// SIMATIC S7-200 project (STEP 7-Micro/WIN), CPU 224 REL 02.01

ORGANIZATION_BLOCK Briquette_Press_B_41:OB1
TITLE=B V4.1
// Custom program for WEIMA TH Standard Series briquette press.
//  #NVJOB Nicholas Veselov (independent developer) - https://nvjob.pro, http://nvjob.dx.am
// 
// ---------------------------------------------------------------------
// 
// INPUTS
// I0.0 - Power.
// I0.1 - Start the program in automatic mode.
// I0.2 - Stop the program in automatic mode.
// I0.3 - Manual mode.
// I0.4 - Vertical piston, sensor, lower position.
// I0.5 - Vertical piston, sensor, upper position.
// I0.6 - Horizontal piston, sensor, position retracted.
// I0.7 - Horizontal piston, sensor, position extended.
// I1.0 - Not involved.
// I1.1 - Valve button.
// I1.2 - Accident, stop.
// I1.3 - Change in operating time of the screw. Min time*.
// I1.4 - Change in the operating time of the screw. Max. time*.
// I1.5 - Not involved.
// 
// ---------------------------------------------------------------------
// 
// OUTPUTS
// Q0.0 - The engine of the hydraulic power station (star-delta).
// Q0.1 - Hydroelectric power station engine (star-delta).
// Q0.2 - Fan.
// Q0.3 - Auger.
// Q0.4 - Vertical piston, valve, up position (pushes down).
// Q0.5 - Vertical piston, valve, lower position (pushes up).
// Q0.6 - Horizontal piston, valve, retracts the piston.
// Q0.7 - Horizontal piston, valve, extends the piston.
// Q1.0 - Collet Piston.
// Q1.1 - Light Bulb Start
// 
BEGIN
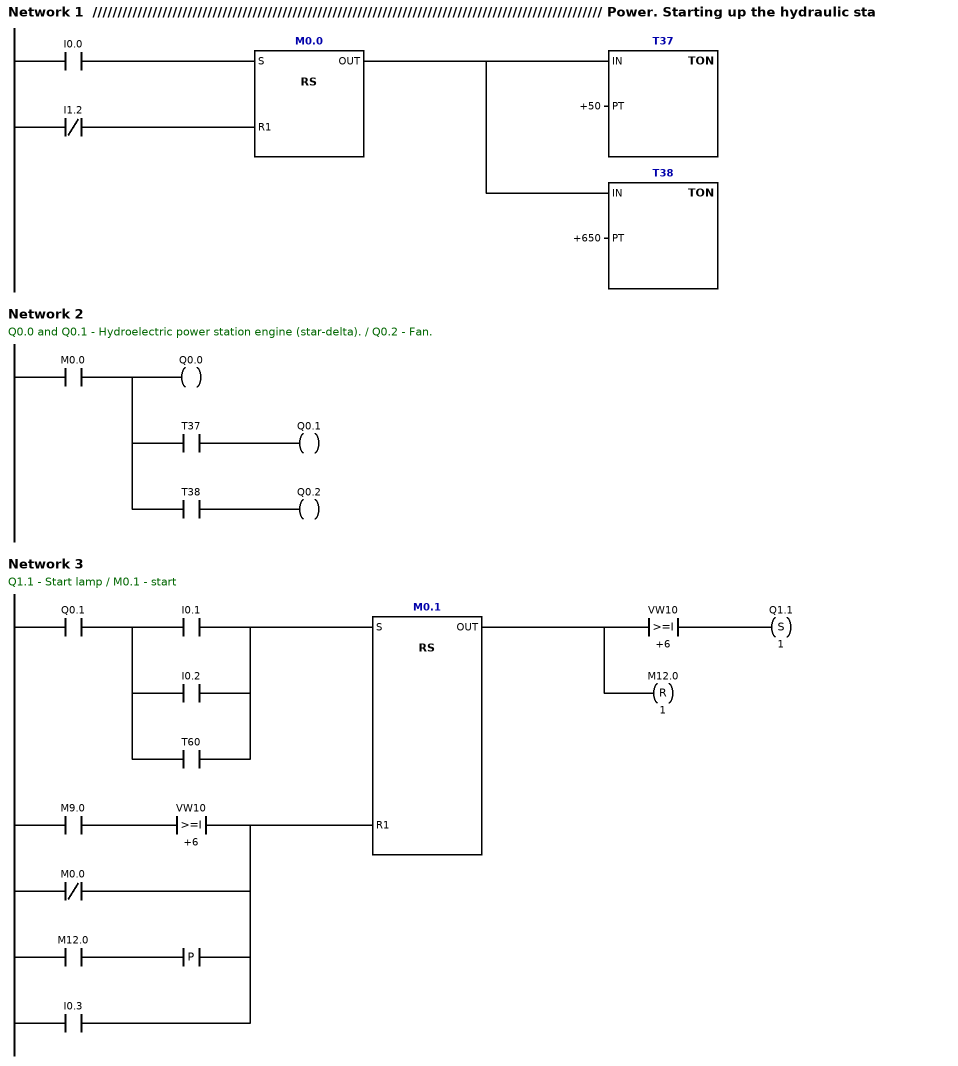
Network 1 // //////////////////////////////////////////////////////////////////////////////////////////////////////
Power. Starting up the hydraulic station.
//////////////////////////////////////////////////////////////////////////////////////////////////////
LD     I0.0
LDN    I1.2
NOT
LPS
A      M0.0
=      M0.0
LPP
ALD
O      M0.0
=      M0.0
TON    T37, +50
TON    T38, +650
Network 2
// Q0.0 and Q0.1 - Hydroelectric power station engine (star-delta).
// Q0.2 - Fan.
LD     M0.0
LPS
=      Q0.0
A      T37
=      Q0.1
LPP
A      T38
=      Q0.2
Network 3
// Q1.1 - Start lamp
// M0.1 - start
// (network saved uncompiled; LAD cells follow)
// row 0: c0 -| |- Q0.1 v  c1 -| |- I0.1 v  c2 --  c3 [RS M0.1 S:=power@row0, R1:=power@row3, OUT=>power]  c4 -- v  c5 -|>=I|- VW10, +6  c6 -(S) Q1.1, 1
// row 1: c0 ^v  c1 -| |- I0.2 ^v  c3 [box]  c4 ^  c5 -(R) M12.0, 1
// row 2: c0 ^  c1 -| |- T60 ^  c3 [box]
// row 3: c0 -| |- M9.0  c1 -|>=I|- VW10, +6 v  c2 --  c3 [box]
// row 4: c0 -|/|- M0.0  c1 -- ^v
// row 5: c0 -| |- M12.0  c1 -|P|-  ^v
// row 6: c0 -| |- I0.3  c1 -- ^
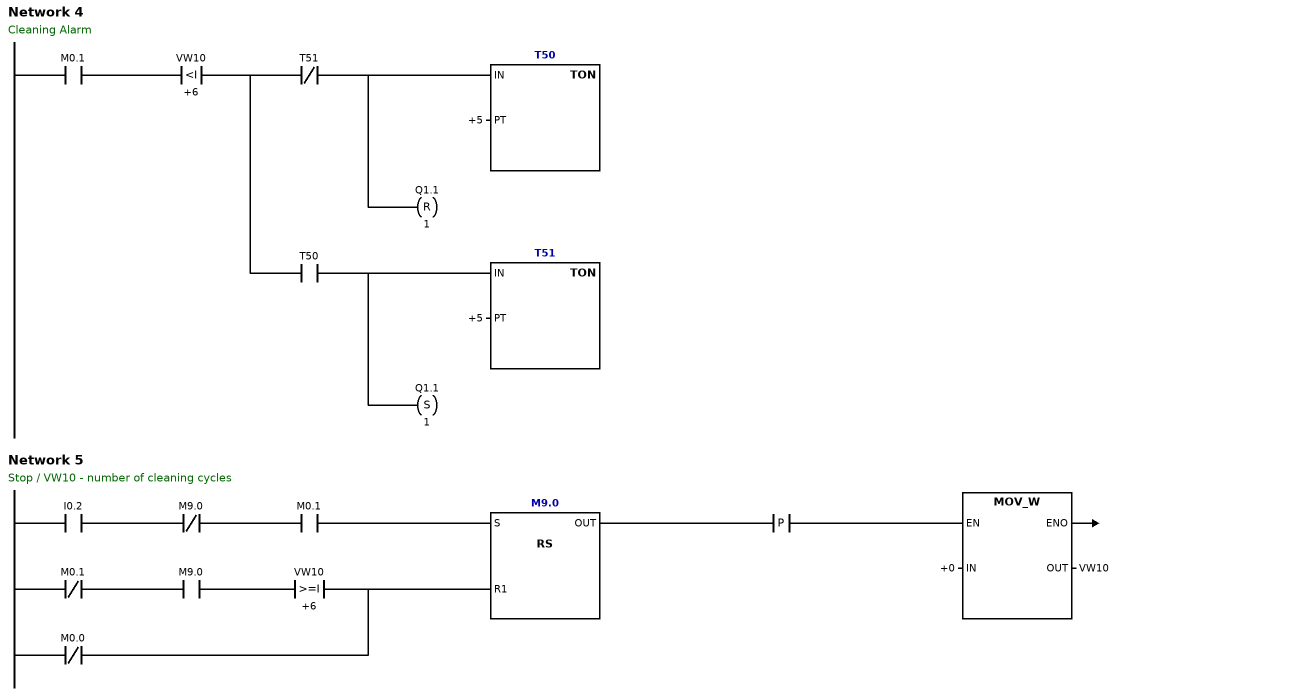
Network 4
// Cleaning Alarm
// (network saved uncompiled; LAD cells follow)
// row 0: c0 -| |- M0.1  c1 -|<I|- VW10, +6 v  c2 -|/|- T51 v  c3 --  c4 [TON T50 IN:=power@row0, PT:=+5]
// row 1: c1 ^v  c2 ^v  c4 [box]
// row 2: c1 ^v  c2 ^  c3 -(R) Q1.1, 1
// row 3: c1 ^  c2 -| |- T50 v  c3 --  c4 [TON T51 IN:=power@row3, PT:=+5]
// row 4: c2 ^v  c4 [box]
// row 5: c2 ^  c3 -(S) Q1.1, 1
Network 5
// Stop
// VW10 - number of cleaning cycles
// (network saved uncompiled; LAD cells follow)
// row 0: c0 -| |- I0.2  c1 -|/|- M9.0  c2 -| |- M0.1  c3 --  c4 [RS M9.0 S:=power@row0, R1:=power@row1, OUT=>power]  c5 --  c6 -|P|-  c7 --  c8 [MOV_W EN:=power@row0, IN:=+0, ENO=>power, OUT=>VW10]  c9 ->
// row 1: c0 -|/|- M0.1  c1 -| |- M9.0  c2 -|>=I|- VW10, +6 v  c3 --  c4 [box]  c8 [box]
// row 2: c0 -|/|- M0.0  c1 --  c2 -- ^
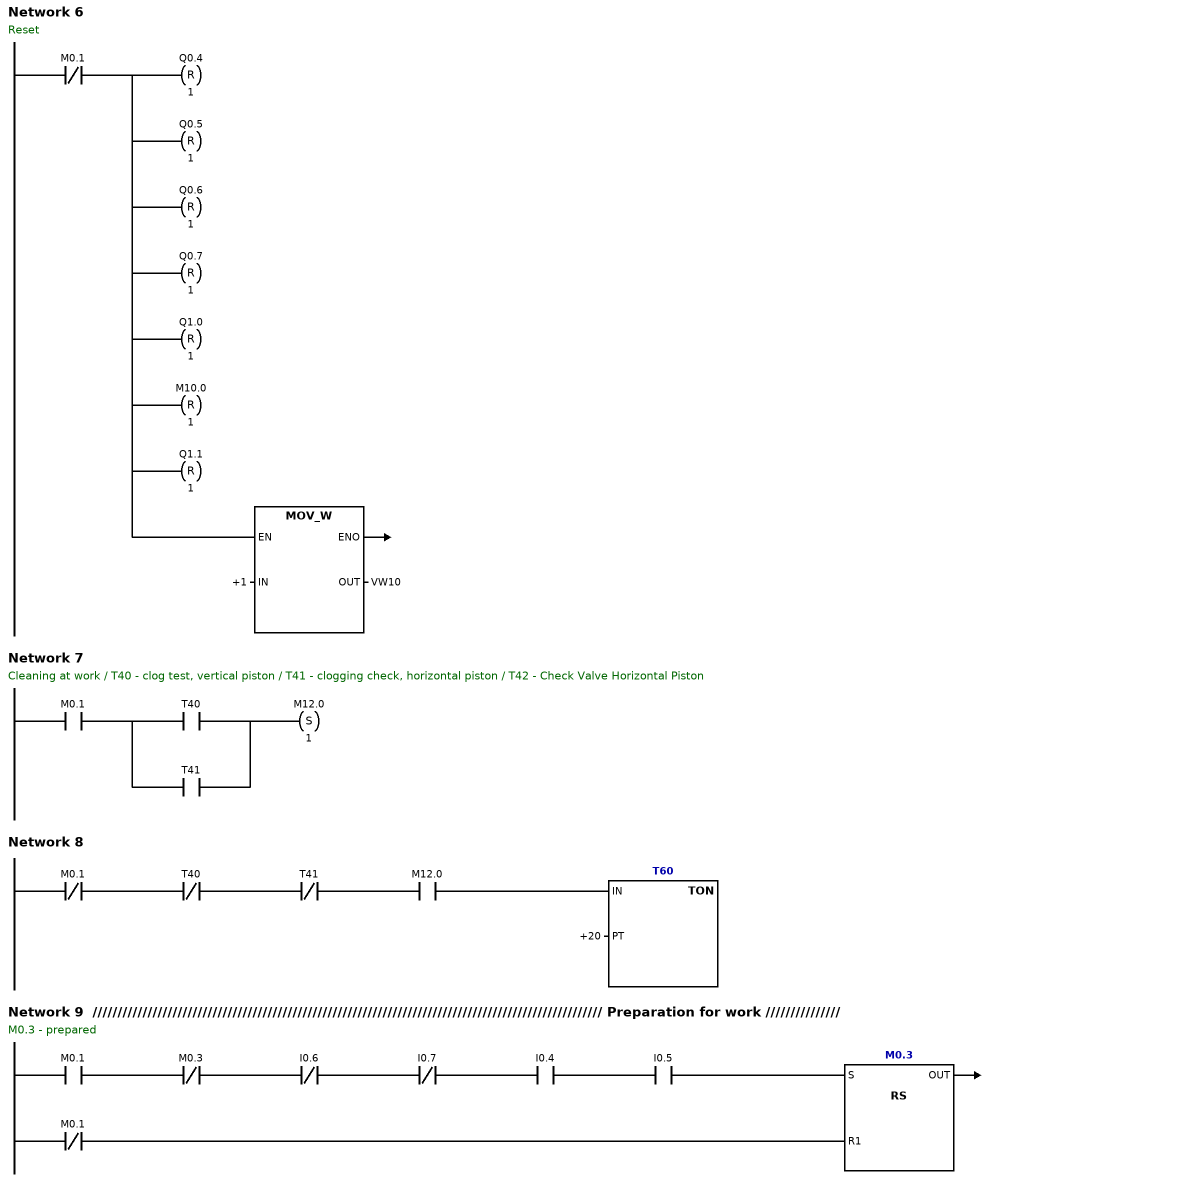
Network 6
// Reset
LDN    M0.1
R      Q0.4, 1
R      Q0.5, 1
R      Q0.6, 1
R      Q0.7, 1
R      Q1.0, 1
R      M10.0, 1
R      Q1.1, 1
MOVW   +1, VW10
Network 7
// Cleaning at work
// T40 - clog test, vertical piston
// T41 - clogging check, horizontal piston
// T42 - Check Valve Horizontal Piston
LD     M0.1
LD     T40
O      T41
ALD
S      M12.0, 1
Network 8
LDN    M0.1
AN     T40
AN     T41
A      M12.0
TON    T60, +20
Network 9 // //////////////////////////////////////////////////////////////////////////////////////////////////////
Preparation for work
//////////////////////////////////////////////////////////////////////////////////////////////////////
// M0.3 - prepared
LD     M0.1
AN     M0.3
AN     I0.6
AN     I0.7
A      I0.4
A      I0.5
LDN    M0.1
NOT
LPS
A      M0.3
=      M0.3
LPP
ALD
O      M0.3
=      M0.3
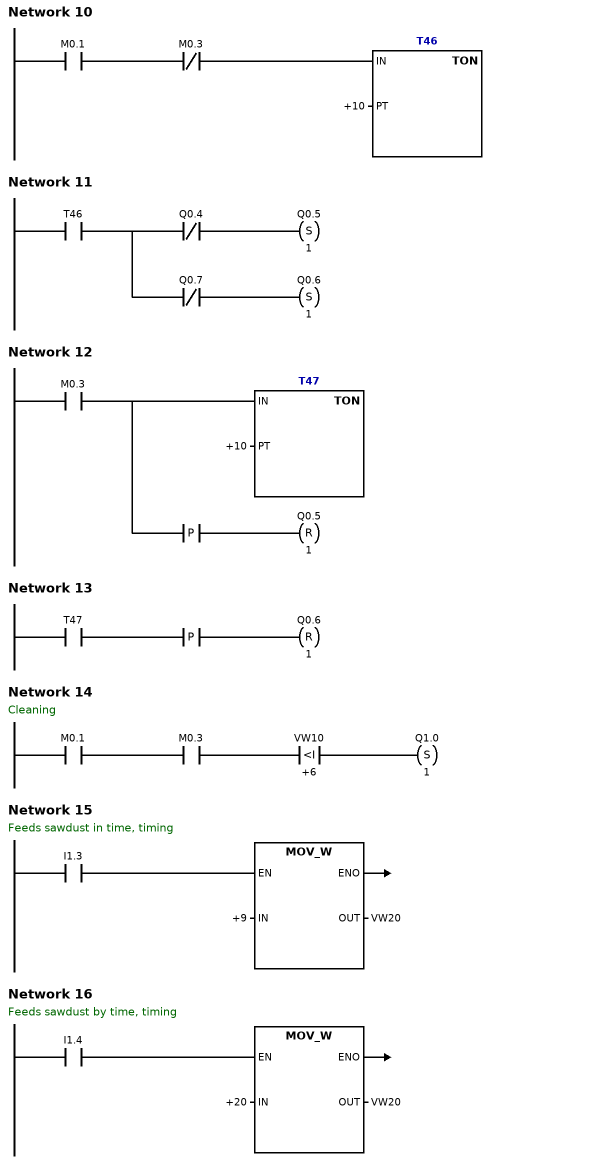
Network 10
LD     M0.1
AN     M0.3
TON    T46, +10
Network 11
LD     T46
LPS
AN     Q0.4
S      Q0.5, 1
LPP
AN     Q0.7
S      Q0.6, 1
Network 12
LD     M0.3
TON    T47, +10
EU
R      Q0.5, 1
Network 13
LD     T47
EU
R      Q0.6, 1
Network 14
// Cleaning
// (network saved uncompiled; LAD cells follow)
// row 0: c0 -| |- M0.1  c1 -| |- M0.3  c2 -|<I|- VW10, +6  c3 -(S) Q1.0, 1
Network 15
// Feeds sawdust in time, timing
LD     I1.3
MOVW   +9, VW20
Network 16
// Feeds sawdust by time, timing
LD     I1.4
MOVW   +20, VW20
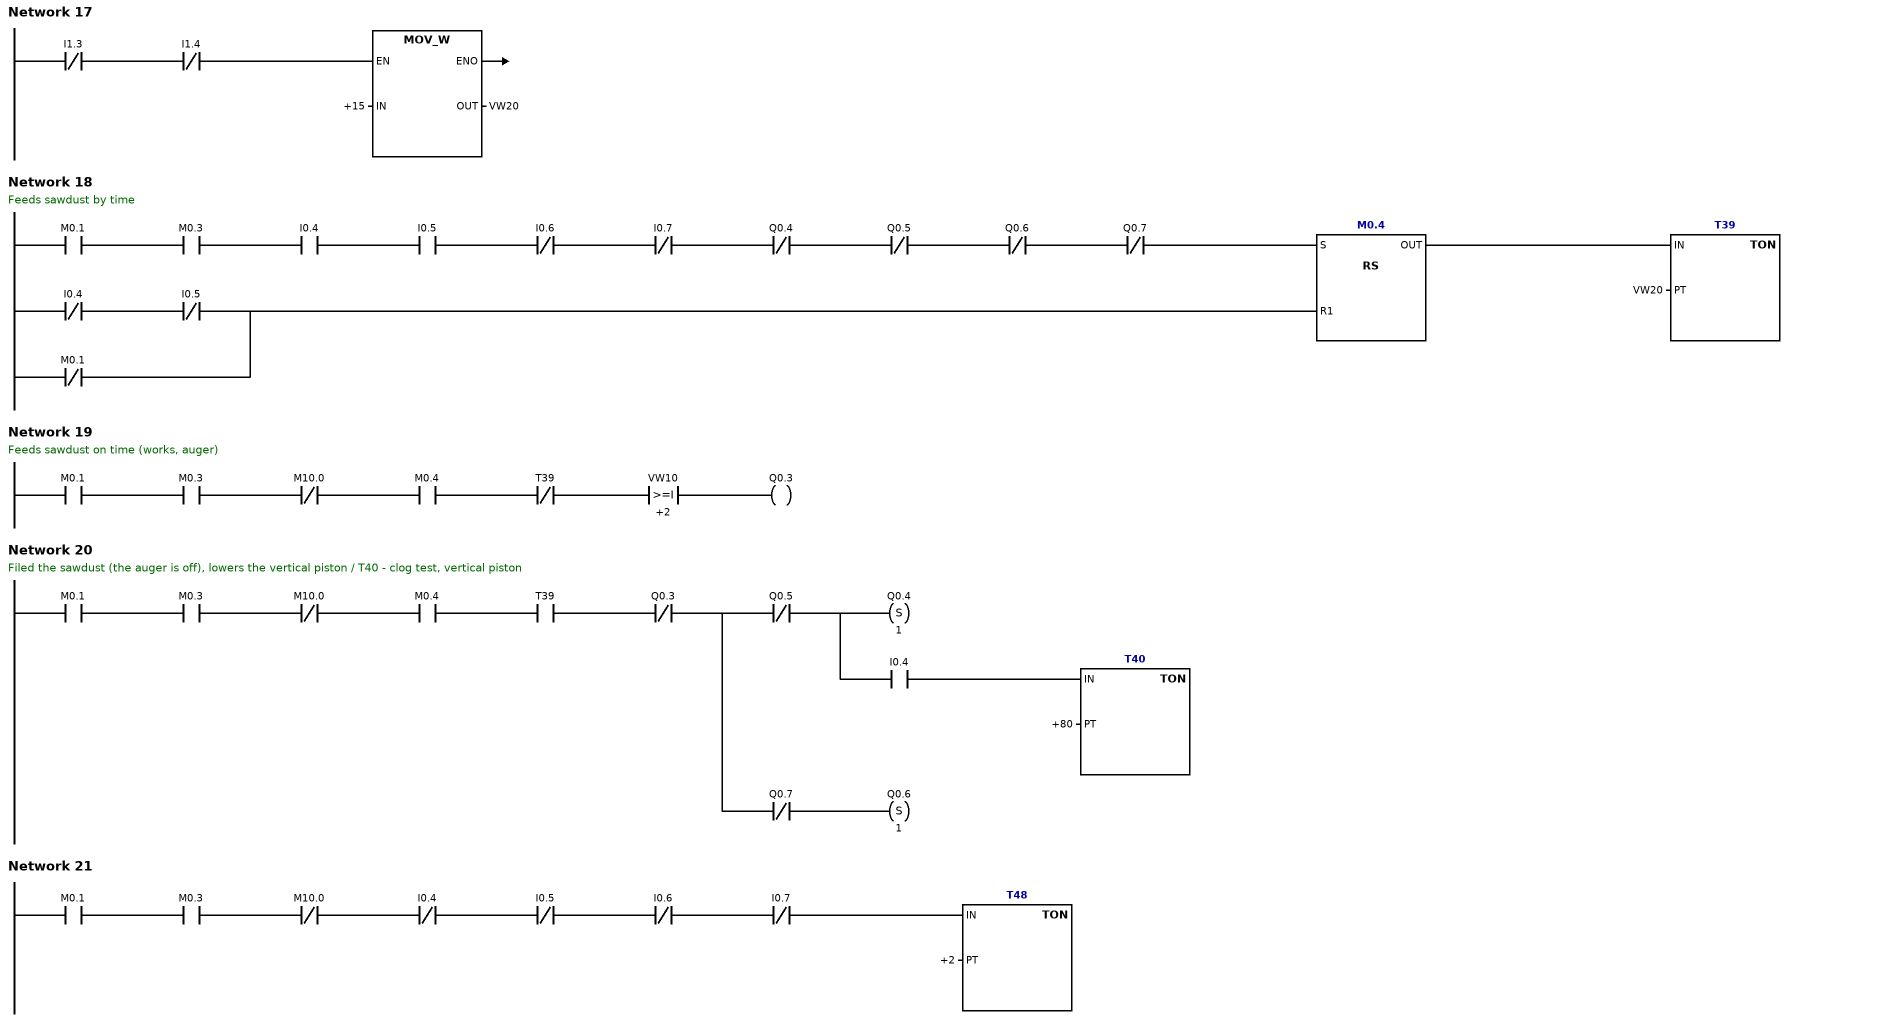
Network 17
LDN    I1.3
AN     I1.4
MOVW   +15, VW20
Network 18
// Feeds sawdust by time
LD     M0.1
A      M0.3
A      I0.4
A      I0.5
AN     I0.6
AN     I0.7
AN     Q0.4
AN     Q0.5
AN     Q0.6
AN     Q0.7
LDN    I0.4
AN     I0.5
ON     M0.1
NOT
LPS
A      M0.4
=      M0.4
LPP
ALD
O      M0.4
=      M0.4
TON    T39, VW20
Network 19
// Feeds sawdust on time (works, auger)
// (network saved uncompiled; LAD cells follow)
// row 0: c0 -| |- M0.1  c1 -| |- M0.3  c2 -|/|- M10.0  c3 -| |- M0.4  c4 -|/|- T39  c5 -|>=I|- VW10, +2  c6 -( ) Q0.3
Network 20
// Filed the sawdust (the auger is off), lowers the vertical piston
// T40 - clog test, vertical piston
LD     M0.1
A      M0.3
AN     M10.0
A      M0.4
A      T39
AN     Q0.3
LPS
AN     Q0.5
S      Q0.4, 1
A      I0.4
TON    T40, +80
LPP
AN     Q0.7
S      Q0.6, 1
Network 21
LD     M0.1
A      M0.3
AN     M10.0
AN     I0.4
AN     I0.5
AN     I0.6
AN     I0.7
TON    T48, +2
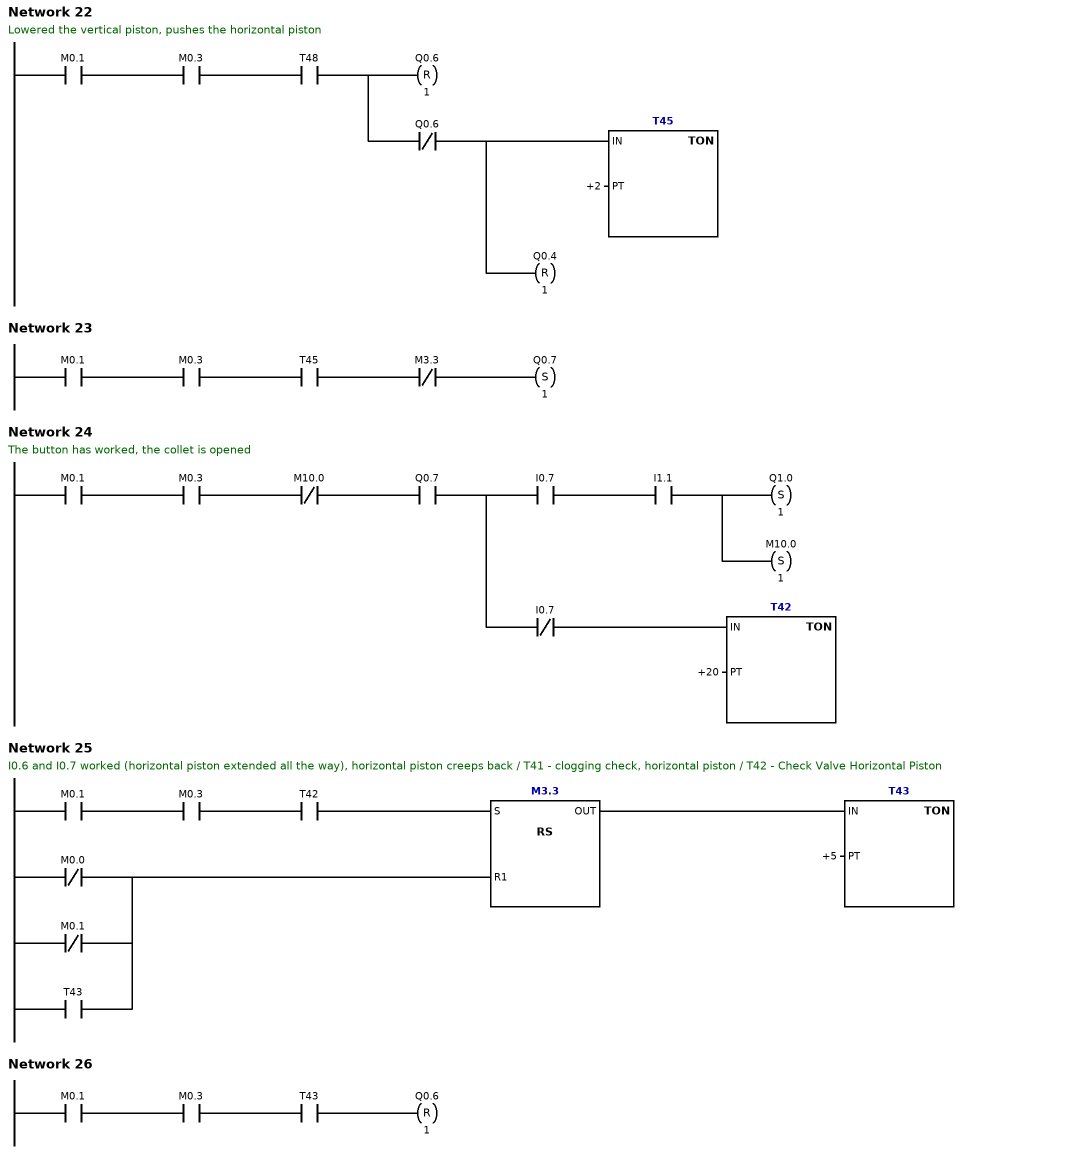
Network 22
// Lowered the vertical piston, pushes the horizontal piston
LD     M0.1
A      M0.3
A      T48
R      Q0.6, 1
AN     Q0.6
TON    T45, +2
R      Q0.4, 1
Network 23
LD     M0.1
A      M0.3
A      T45
AN     M3.3
S      Q0.7, 1
Network 24
// The button has worked, the collet is opened
LD     M0.1
A      M0.3
AN     M10.0
A      Q0.7
LPS
A      I0.7
A      I1.1
S      Q1.0, 1
S      M10.0, 1
LPP
AN     I0.7
TON    T42, +20
Network 25
// I0.6 and I0.7 worked (horizontal piston extended all the way), horizontal piston creeps back
// T41 - clogging check, horizontal piston
// T42 - Check Valve Horizontal Piston
LD     M0.1
A      M0.3
A      T42
LDN    M0.0
ON     M0.1
O      T43
NOT
LPS
A      M3.3
=      M3.3
LPP
ALD
O      M3.3
=      M3.3
TON    T43, +5
Network 26
LD     M0.1
A      M0.3
A      T43
R      Q0.6, 1
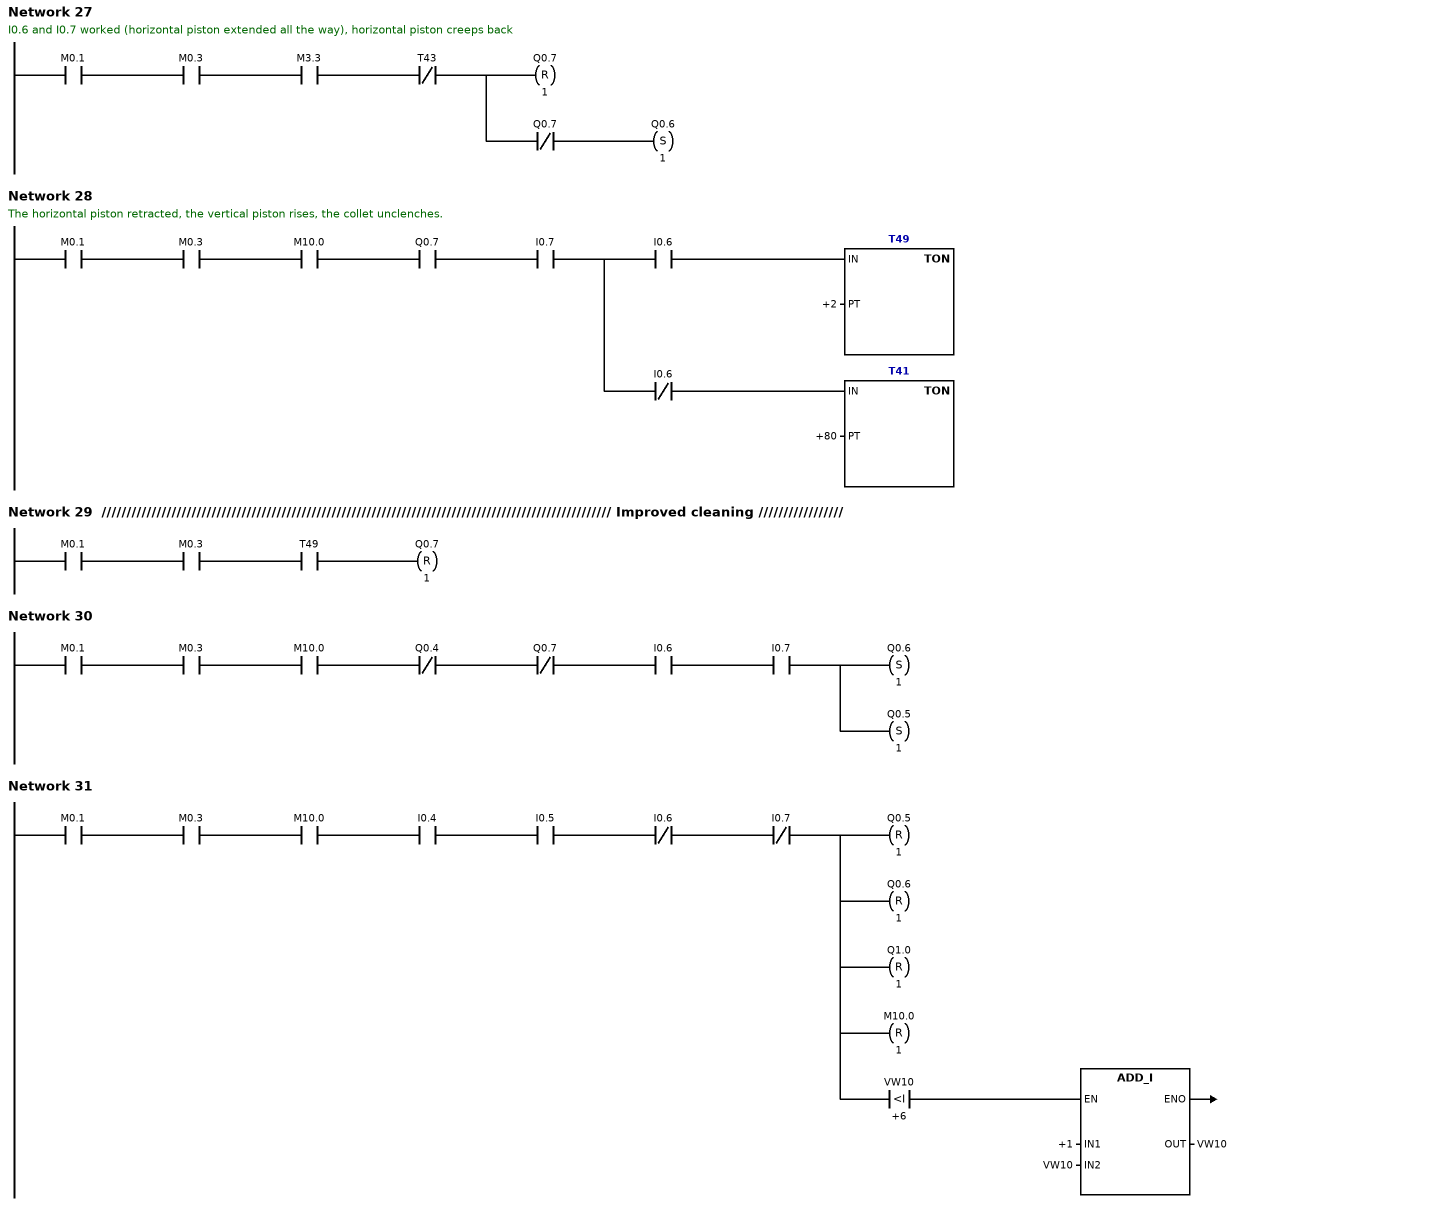
Network 27
// I0.6 and I0.7 worked (horizontal piston extended all the way), horizontal piston creeps back
LD     M0.1
A      M0.3
A      M3.3
AN     T43
R      Q0.7, 1
AN     Q0.7
S      Q0.6, 1
Network 28
// The horizontal piston retracted, the vertical piston rises, the collet unclenches.
LD     M0.1
A      M0.3
A      M10.0
A      Q0.7
A      I0.7
LPS
A      I0.6
TON    T49, +2
LPP
AN     I0.6
TON    T41, +80
Network 29 // //////////////////////////////////////////////////////////////////////////////////////////////////////
Improved cleaning
//////////////////////////////////////////////////////////////////////////////////////////////////////
LD     M0.1
A      M0.3
A      T49
R      Q0.7, 1
Network 30
LD     M0.1
A      M0.3
A      M10.0
AN     Q0.4
AN     Q0.7
A      I0.6
A      I0.7
S      Q0.6, 1
S      Q0.5, 1
Network 31
// (network saved uncompiled; LAD cells follow)
// row 0: c0 -| |- M0.1  c1 -| |- M0.3  c2 -| |- M10.0  c3 -| |- I0.4  c4 -| |- I0.5  c5 -|/|- I0.6  c6 -|/|- I0.7 v  c7 -(R) Q0.5, 1
// row 1: c6 ^v  c7 -(R) Q0.6, 1
// row 2: c6 ^v  c7 -(R) Q1.0, 1
// row 3: c6 ^v  c7 -(R) M10.0, 1
// row 4: c6 ^  c7 -|<I|- VW10, +6  c8 --  c9 [ADD_I EN:=power@row4, IN1:=+1, IN2:=VW10, ENO=>power, OUT=>VW10]  c10 ->
// row 5: c9 [box]
END_ORGANIZATION_BLOCK
